(* PLC project LibIT_SYS, lamsystems-it.ru LibIT_SYS 1 *)
(* stored: creationDateTime 2020-10-15T08:18:12, productRelease 0, modificationDateTime 2020-10-15T08:26:49, version 1 *)

(* Программная перезагрузка устройства *)
FUNCTION SoftReset : BOOL
  VAR_INPUT
    Ex : BOOL := FALSE;  (* Разрешение исполнения *)
  END_VAR

            {extern void AppSys_SoftReset(BOOL);AppSys_SoftReset(EX);}
SoftReset:= TRUE;

          
END_FUNCTION
